TYPE tyRampOutputs :
STRUCT
bRampActivated: BOOL ; 	
iRampValueOutput : INT ; 
iCurrentStep :INT ; 
bRampDone : BOOL;
dwError: ARRAY[0..10] OF BOOL; ; 
END_STRUCT
END_TYPE

(* stored: Version 1.1.0.1
   DUT tyRampOutputs: Id {c4367998-865c-44a0-ac7b-aa502212af99} *)
